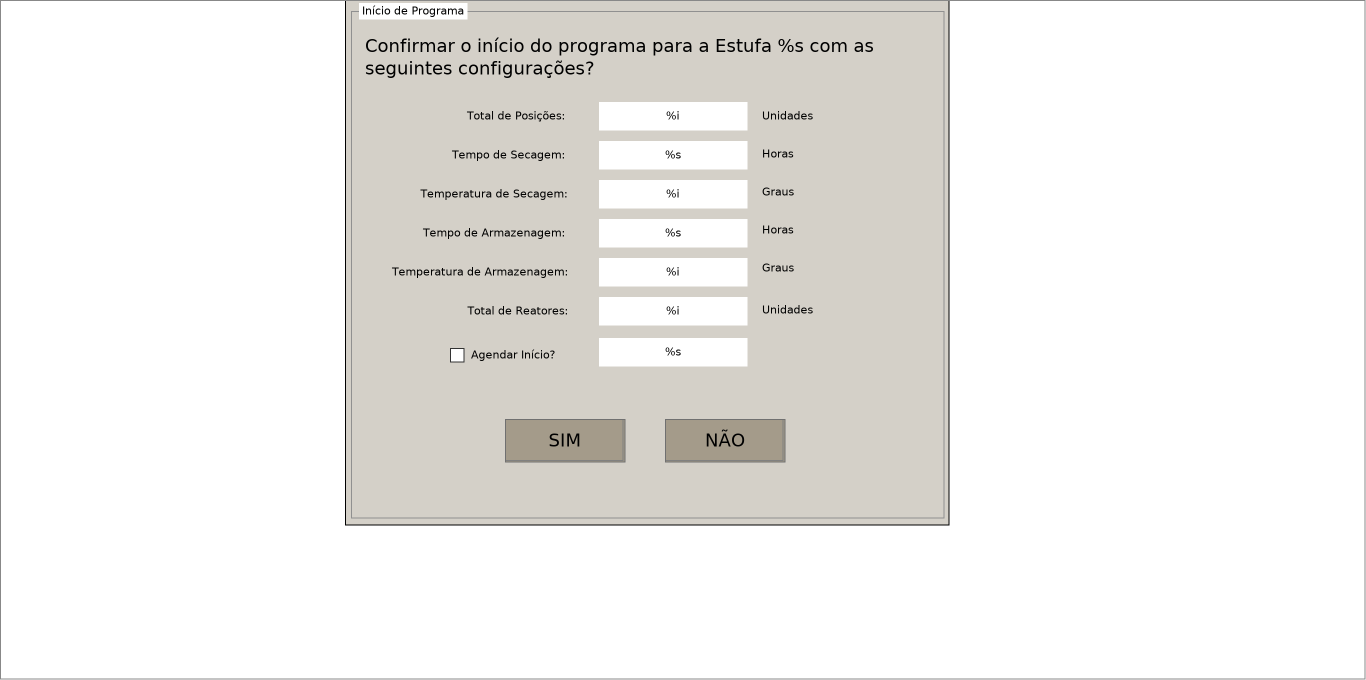
VISUALIZATION IniciaProg_2  // 1366x680
    Rectangle (345,0 604x525)
    GroupBox (351,3 593x515), "Início de Programa"
        Label (111,98 108x30), "Total de Posições:"
        Textfield (247,98 150x30), "%i", text variable: GVL.totalPos[GVL.actEst]
        Label (99,137 117x30), "Tempo de Secagem:"
        Label (65,176 156x30), "Temperatura de Secagem:"
        Label (67,215 152x30), "Tempo de Armazenagem:"
        Label (37,254 184x30), "Temperatura de Armazenagem:"
        Label (113,293 108x30), "Total de Reatores:"
        Textfield (247,137 150x30), "%s", text variable: GVL.totalSeca[GVL.actEst]
        Textfield (247,176 150x30), "%i", text variable: GVL_P.arrStatusEstufas[gvl.actEst].tempSeca
        Textfield (247,215 150x30), "%s", text variable: GVL.totalArm[GVL.actEst]
        Textfield (247,254 150x30), "%i", text variable: GVL_P.arrStatusEstufas[gvl.actEst].tempArm
        Textfield (247,293 150x30), "%i", text variable: GVL.totalRaet[GVL.actEst]
        Label (408,98 62x30), "Unidades"
        Label (408,136 62x30), "Horas"
        Label (408,174 62x30), "Graus"
        Label (408,212 62x30), "Horas"
        Label (408,250 62x30), "Graus"
        Label (408,292 62x30), "Unidades"
        Button (154,416 120x43), "SIM"
            OnMouseClick: CloseDialog Dialog=IniciaProg_2, Result=Yes, NumpadKeypadSet=True
            OnMouseClick: execute { simIniciaProg(); }
        Button (314,416 120x43), "NÃO"
            OnMouseClick: CloseDialog Dialog=IniciaProg_2, Result=No, NumpadKeypadSet=True
        Textfield (247,334 150x30), "%s", text variable: GVL.progInicio[GVL.actEst], input disabled if: not GVL.bAgendaInicio
            OnMouseClick: OpenDialog Dialog=setInicio, OpenModal=True, OpenCentered=True
            OnMouseClick: execute {
                gvl.dia:= MID(STR:= gvl.progInicio[gvl.actEst] , LEN:= 2, POS:=12);
                gvl.mes:= MID(STR:= gvl.progInicio[gvl.actEst] , LEN:= 2, POS:=9);
                gvl.ano:= MID(STR:= gvl.progInicio[gvl.actEst] , LEN:= 2, POS:=6);
                gvl.hora:= MID(STR:= gvl.progInicio[gvl.actEst] , LEN:= 2, POS:=15);
                gvl.minuto:= MID(STR:= gvl.progInicio[gvl.actEst] , LEN:= 2, POS:=18);
            }
    Checkbox (448,341 122x28), "Agendar Início?", variable: GVL.bAgendaInicio
    Rectangle (362,30 574x54), "Confirmar o início do programa para a Estufa %s com as seguintes configurações?", text variable: GVL.estAtiva
END_VISUALIZATION

(* stored: Version 1.1.0.1, ProductVersion 3.1.4024.12
   Visu IniciaProg_2: Id {c2645cd2-587d-43dd-b3f4-cff6734f5470} *)
